(* IEC 61131-3 sources: SmartHomeNew/snapshots/project_clean_state_2026_04_16/workspace/dut_rebuild/lighting_v2/extraction, 1 file *)

(* ---- FB_Lighting_Command_Extractor_DRAFT.st ---- *)
FUNCTION_BLOCK FB_Lighting_Command_Extractor_DRAFT
VAR_INPUT
    VI_Enable : BOOL;
    VI_Brightness_Setpoint : REAL;
END_VAR
VAR_OUTPUT
    VO_Command : ST_Lighting_Command_V2;
END_VAR

VO_Command.Enabled := VI_Enable;
VO_Command.Brightness_Setpoint := VI_Brightness_Setpoint;
END_FUNCTION_BLOCK
